(* IEC 61131-3 sources: Palletizer_Control_with_Automation_Studio/Task_2/Logical/PLCopen, 3 files *)

(* ---- Types.typ ---- *)
TYPE
	State_type :
		(
		IDLE,
		ENABLE_AXES,
		BELT_MOVING,
		BELT_STOPPING,
		BELT_HOLDING,
		CUTTER_BACK,
		CUTTER_END
		);
END_TYPE

(* ---- Main.st ---- *)
PROGRAM _INIT
	(* Insert code here *)

END_PROGRAM

PROGRAM _CYCLIC
	Enable := TRUE;

	IF STOP THEN
		CutterEnable := FALSE;
		ConveyorEnable := FALSE;

		Cutter.AxisCommand := AXIS_STOP;
		Conveyor.AxisCommand := MOVE_ADDITIVE;
		Conveyor.AxisCommand := AXIS_STOP;

		Stop_Light := TRUE;
		Green_Light := FALSE;
		White_Light := FALSE;
		Yellow_Light := FALSE;

		State := IDLE;
	END_IF

	CASE State OF
		IDLE:
			IF START_BUTTON THEN
				CutterEnable := TRUE;
				ConveyorEnable := TRUE;

				Cutter.AxisCommand := AXIS_STOP;
				Conveyor.AxisCommand := AXIS_STOP;

				Stop_Light := FALSE;
				Green_Light := TRUE;
				White_Light := FALSE;
				Yellow_Light := FALSE;

				State := ENABLE_AXES;
			END_IF

		ENABLE_AXES:
			IF Cutter.Status = STANDSTILL AND Conveyor.Status = STANDSTILL THEN
				Conveyor.AxisCommand := MOVE_VELOCITY;

				Stop_Light := FALSE;
				Green_Light := TRUE;
				White_Light := TRUE;
				Yellow_Light := FALSE;

				State := BELT_MOVING;
			END_IF

		BELT_MOVING:
			IF TRIGGER_INPUT THEN
				Conveyor.AxisCommand := MOVE_ADDITIVE;

				State := BELT_STOPPING;
			END_IF

		BELT_STOPPING:
			IF Conveyor.CommandExecuted THEN
				Conveyor.AxisCommand := AXIS_STOP;
				Cutter.AxisCommand := MOVE_ADDITIVE;
				Cutter.Position := CUTTER_END_POSE;

				Stop_Light := FALSE;
				Green_Light := TRUE;
				White_Light := FALSE;
				Yellow_Light := TRUE;

				State := BELT_HOLDING;
			END_IF

		BELT_HOLDING:
			IF Cutter.CommandExecuted THEN
				Cutter.AxisCommand := AXIS_STOP;

				State := CUTTER_BACK;
			END_IF

		CUTTER_BACK:
			IF NOT Cutter.CommandExecuted THEN
				Cutter.AxisCommand := MOVE_ADDITIVE;
				Cutter.Position := -CUTTER_END_POSE;

				State := CUTTER_END;
			END_IF

		CUTTER_END:
			IF Cutter.CommandExecuted THEN
				Cutter.AxisCommand := AXIS_STOP;

				State := ENABLE_AXES;
			END_IF
	END_CASE

	Conveyor.Slave := ADR(gAxis01);
	Conveyor.Position := 2*BELT_DISTANCE;
	Conveyor.Velocity := velocity;
	Conveyor.Acceleration := 100;
	Conveyor.Deceleration := 100;

	Conveyor(AxisEnable := ConveyorEnable);
	ConveyorPosition := Conveyor.ActualPosition;

	Cutter.Slave := ADR(gAxis02);
	Cutter.Velocity := CUTTER_SPEED;
	Cutter.Acceleration := 100;
	Cutter.Deceleration := 100;

	Cutter(AxisEnable := CutterEnable);
	CutterPosition := Cutter.ActualPosition;

END_PROGRAM

PROGRAM _EXIT
	(* Insert code here *)

END_PROGRAM

(* ---- Variables.var ---- *)
VAR
	State : State_type;
	GA_test : GenericAxis_FB;
	velocity : REAL := 100;
	ConveyorEnable : BOOL;
	CutterEnable : BOOL;
	Enable : BOOL;
	result : INT;
	Command : WORD := MOVE_VELOCITY;
	Actuation : INT;
	Cutter : GenericAxis_FB;
	Conveyor : GenericAxis_FB;
END_VAR
